// TIA Portal V20 export
// export: Created 2026-08-17T22:42:35.4751908Z, ExportSetting None, DisplayName Totally Integrated Automation Portal, DisplayVersion V20 Update 3, DisplayName TIA Portal Openness, DisplayVersion V20 Update 3, DisplayName TIA Portal Version Control Interface, DisplayVersion V20 Update 3, DisplayName STEP 7 Professional, DisplayVersion V20 Update 3, DisplayName STEP 7 Safety, DisplayVersion V20 Update 2, DisplayName WinCC Basic/Comfort/Advanced, DisplayVersion V20 Update 3, DisplayName SIMATIC Visualization Architect, DisplayVersion V20 Update 3, DisplayName WinCC Unified, DisplayVersion V20 Update 3, DisplayName SIMATIC Visualization Architect, DisplayVersion V20 Update 3
FUNCTION_BLOCK "EM_Inlet"   // FB20, LAD
{ S7_Optimized_Access := 'TRUE' }
// stored: MemoryReserve 100, SetENOAutomatically false
   VAR
      ValveA { S7_SetPoint := 'True'} : "Valve2Coil";
   END_VAR
BEGIN

REGION Network 1: Valve A -
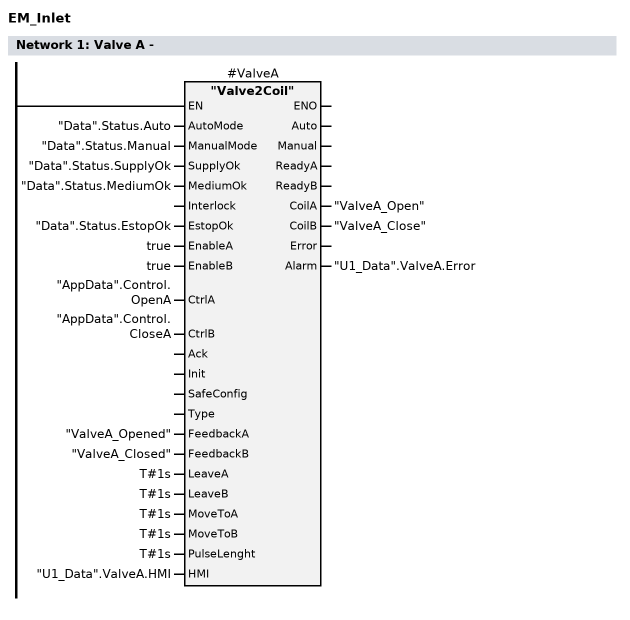
   RUNG wire#powerrail
      #ValveA(AutoMode := "Data".Status.Auto, ManualMode := "Data".Status.Manual, SupplyOk := "Data".Status.SupplyOk, MediumOk := "Data".Status.MediumOk, Interlock :=, EstopOk := "Data".Status.EstopOk, EnableA := true, EnableB := true, CtrlA := "AppData".Control.OpenA, CtrlB := "AppData".Control.CloseA, Ack :=, Init :=, SafeConfig :=, "Type" :=, FeedbackA := "ValveA_Opened", FeedbackB := "ValveA_Closed", LeaveA := T#1s, LeaveB := T#1s, MoveToA := T#1s, MoveToB := T#1s, PulseLenght := T#1s, HMI := "U1_Data".ValveA.HMI, Auto =>, Manual =>, ReadyA =>, ReadyB =>, CoilA => "ValveA_Open", CoilB => "ValveA_Close", Error =>, Alarm => "U1_Data".ValveA.Error)
   END_RUNG
   // the same network as SCL:
   #ValveA(AutoMode := "Data".Status.Auto,   // "Valve2Coil"
           ManualMode := "Data".Status.Manual,
           SupplyOk := "Data".Status.SupplyOk,
           MediumOk := "Data".Status.MediumOk,
           EstopOk := "Data".Status.EstopOk,
           EnableA := true,
           EnableB := true,
           CtrlA := "AppData".Control.OpenA,
           CtrlB := "AppData".Control.CloseA,
           FeedbackA := "ValveA_Opened",
           FeedbackB := "ValveA_Closed",
           LeaveA := T#1s,
           LeaveB := T#1s,
           MoveToA := T#1s,
           MoveToB := T#1s,
           PulseLenght := T#1s,
           HMI := "U1_Data".ValveA.HMI,
           CoilA => "ValveA_Open",
           CoilB => "ValveA_Close",
           Alarm => "U1_Data".ValveA.Error);
END_REGION
END_FUNCTION_BLOCK
